// Mitsubishi GX Works2 project: 펄스셋리셋   PLC: Q02/Q02H

PROGRAM MAIN
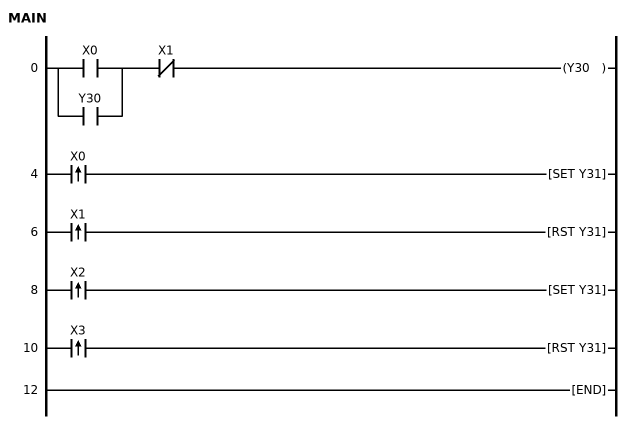
0     LD      X0
      OR      Y30
      ANI     X1
      OUT     Y30
4     LDP     X0
      SET     Y31
6     LDP     X1
      RST     Y31
8     LDP     X2
      SET     Y31
10    LDP     X3
      RST     Y31
12    END
END_PROGRAM
